// TIA Portal V19 export
Connection "HMI_Connection_1"  Driver=SMART_S7_1200_OMS, InterfaceType=ETHERNET, PhysicId=S7_ETHERNET_IP4, ProtocolId=S7_ETHERNET_IP4
  NameValuePair "LocAddress"  Value=192.168.0.2
  NameValuePair "RemStAddress"  Value=192.168.0.1
